FUNCTION_BLOCK ABSTRACT ReadyProgramState EXTENDS ProgramState

{attribute 'monitoring' := 'call'}
{attribute 'OPC.UA.DA.Property' := '1'}
{attribute 'OPC.UA.DA.Access' := '1'}
PROPERTY FINAL Name : STRING
GET
Name := 'Ready';
END_GET
END_PROPERTY

END_FUNCTION_BLOCK

(* stored: Version 1.1.0.1
   POU ReadyProgramState: Id {a809a80e-4ede-428a-bcc8-804e808d41fe}, SpecialFunc None
   Property Name: Id {2eafe4a6-8d61-4fbc-8e35-2d7997fb97f6}
   Get Get: Id {8d0105fe-43f6-483a-b829-b6f743afeeb4} *)
